ABB RobotStudio station: Station_[09.05.13]workingpinattach.rspag

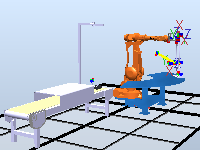
--- station ---
Station Station_[09.05.13]workingpinattach (saved by RobotStudio format 3)
Controller IRB2400_10kg_1.5m_3, task T_ROB1: task frame (RAPID world) sits at (0, 0, 226) mm in the station
Controller IRB2400_10kg_1.5m_3
  mechanical unit ROB_1: IRB2400_10_150__02, 6 joints, base frame (0, 0, -10) mm
Layout (positions relative to the parent item):
  - IRB2400_10_150__02 [mechanism, from Robots\IRB2400_10_150__02.rslib] at (0, 0, 216) mm; joint values [0, 0, 0, 0, 0, 0] (rad or m)
  - Table3_2 [part]
  - SC_RightDispenser [smart component] at (848.89, 660.39, 707) mm, rotated rx 0 ry 0 rz -142.5 deg
      signals: DI diNewPin, DO doPinInPosition2, DO doPinInPosition1
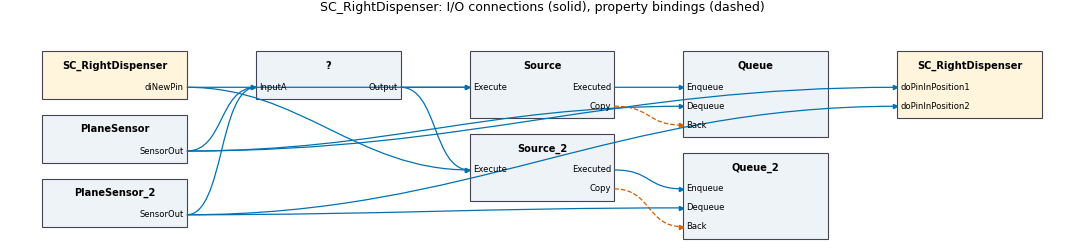
      connections:
        SC_RightDispenser.diNewPin -> Source.Execute
        Source.Executed -> Queue.Enqueue
        PlaneSensor.SensorOut -> Queue.Dequeue
        PlaneSensor.SensorOut -> SC_RightDispenser.doPinInPosition1
        PlaneSensor.SensorOut -> ?.InputA
        ?.Output -> Source.Execute
        SC_RightDispenser.diNewPin -> Source_2.Execute
        Source_2.Executed -> Queue_2.Enqueue
        PlaneSensor_2.SensorOut -> Queue_2.Dequeue
        PlaneSensor_2.SensorOut -> SC_RightDispenser.doPinInPosition2
        PlaneSensor_2.SensorOut -> ?.InputA
        ?.Output -> Source_2.Execute
        Source.Copy => Queue.Back
        Source_2.Copy => Queue_2.Back
    - Dispenser [part]
    - Source [smart component]
        properties: Source=Pin; Copy=Pin_23; Parent=(none); Position=[-0.078 0.0985 0.189]; Orientation=[0 0 0]; Transient=false
        signals: DI Execute, DO Executed
    - Queue [smart component]
        properties: Back=Pin_23; Front=(none); Queue={5aa4b278-0833-4ca9-af8d-253aa8523874};{1baac950-fc54-4ea7-852c-7f888843f6f9};{b4b16473-bd2b-40f5-a110-90fbcba822d9};{d003a69b-5307-4c56-b226-d498155ba824};{d659394f-77c7-41ee-9797-cd61472f6401};{a8294731-aa9f-4324-81a7-55ebbef1ff1c};{1eff712e-2c63-4fa8-99b0-fad1482486d3};{b15f9735-19cd-4f7a-8d4f-e540a16427f5};{02485707-3f80-4cc3-94a6-af0fe382acfb};{ec0e8ce0-b480-4ff5-b740-0a7d244ffb35};{21e78636-7eb3-4061-8dde-926c3e464303};{0772fef3-b80e-464b-9cad-322a585d167a};{d8ed8ead-e522-4938-9c7c-7997e1d5aae1};{4dfefca0-2913-4484-9455-684dfc1cbf5a};{f8c8569f-a97f-4f57-84f0-3da59c0f2755};{9fd95979-e5cf-4fa7-b177-2c560699c82c};{84f56170-3294-4345-a728-b2bfe69be833};{b3710d51-6f0f-48ac-9b0f-811ac7c7d083};{c8300349-23e3-4531-beb4-4210900096fb};{31c2e06e-432b-4cd5-8dfd-12cdd0c38bbf};{f6bc1e00-ec05-46bf-9f1a-fcc25cb6084b};{46f4262a-e9c9-45b1-8eff-bed77a1a9e5b};{07cc3b07-c3da-44db-b33b-99881492d9cc};{0c369fdb-a0e7-4beb-a0c1-abd25c6b2a43};{d9cb4cdb-12a7-4146-bf1e-65335fe6fd56};{f09a15e7-f9e4-4c16-add7-657cccb8590f};{c20793dd-1a91-48a1-8edb-9b1aca8d6d7f};{7fbcc782-7f9e-47c5-a7b7-ac04b253ef72};{f46b459a-9e88-46de-a41f-ecde2c97a1c4};{a4b9086d-e076-476d-b3ee-a23e91ee6609};{9ff53e84-8ebc-4345-9cc4-0476dc4b857f};{650503f2-9794-4bb9-bd75-77f7f6044b7b};{58395fe3-f9e1-4cbe-aa54-a35298f9d1c5};{7826030e-95bb-4bf6-b21f-9a7d91df32f4};{2942a0d1-30e6-4527-84a4-878f9b334dec};{a0ef5e72-34a5-445e-b23b-6c91bdee101a};{aa2624ab-89f7-405f-9ffa-69efbc3a4434};{9792617b-04a4-4cec-aa8d-3159fcd6b685}; NumberOfObjects=0
        signals: DI Enqueue, DI Dequeue, DI Clear, DI Delete, DI DeleteAll
    - LinearMover [smart component]
        properties: Object=Queue; Direction=[0 0 -0.07]; Speed=0.05; Reference=Global; ReferenceObject=(none)
        signals: DI Execute
    - PlaneSensor [smart component]
        properties: Origin=[-0.0530000000000006 0.1235 0.1195]; Axis1=[-0.03 0 0]; Axis2=[0 -0.04 0]; SensedPart=(none)
        signals: DI Active, DO SensorOut
      - _sensorPart_ [part]
    - Pin [part] at (-78, 98.5, 189) mm
    - Source_2 [smart component]
        properties: Source=Pin_2; Copy=Pin_2_24; Parent=(none); Position=[-0.078 -0.0985 0.198]; Orientation=[0 0 0]; Transient=false
        signals: DI Execute, DO Executed
    - Queue_2 [smart component]
        properties: Back=Pin_2_24; Front=(none); Queue={168b000f-829e-439e-a2b5-5bc5735400ce};{aacdfd62-2178-4132-b345-2cd6db76197d};{33bd895a-7dcf-445c-8a77-0a7b01e583dc};{c1a42cbc-38c3-48e5-a615-b149ac9d8780};{fcea76f5-b349-47ef-a520-1d1e9307533b};{d936eec8-07d3-4a18-b33b-be549f4009da};{161ff837-8ce6-447d-8217-59dc5e5add53};{a4db4600-beb4-451b-b75b-f36278185638};{fac26080-080b-42e5-8e31-79509598499f};{631b6ef4-884c-4e99-a73e-a0a20b005bbd};{c6922cb5-858b-4dce-bc49-d50c5bb6ff29};{df2a1232-f236-477f-a341-c0e7247ec374};{648e1593-9b95-4c8f-9a3a-4728290fef8c};{9aba8fcf-9d7f-441d-92fe-144ce1ccaea8};{d7b75440-58f5-4476-b5ce-f36666ff7cde};{5c9701ab-d039-4b3a-b377-62889d6251d5};{ccb0f00a-3f08-42c3-ae08-1f0b770d0277};{706e7c72-34ce-4f8c-bd75-a496f5af5a3b};{9b14f38f-1dc8-4293-b5b1-19b5e9014979};{c981c30e-2b93-423a-a409-ef6430437ced};{65c45e0e-b128-4bcf-862a-bd4cb12c0043};{fb18c748-94d3-4804-ba03-343ec976cce9};{90ce3d6b-e0db-4966-a4a1-dfc91785cb07};{f4c8c46d-6357-42e6-99c9-4a127ac338b9};{b14c1a72-e7b7-41f2-882c-7b7c624fc3bd};{c197bb96-9f99-45e2-aeb0-6d90c68a8177}; NumberOfObjects=0
        signals: DI Enqueue, DI Dequeue, DI Clear, DI Delete, DI DeleteAll
    - LinearMover_2 [smart component]
        properties: Object=Queue_2; Direction=[0 0 -0.07]; Speed=0.05; Reference=Global; ReferenceObject=(none)
        signals: DI Execute
    - PlaneSensor_2 [smart component]
        properties: Origin=[-0.053 -0.1235 0.1195]; Axis1=[-0.03 0 0]; Axis2=[0 0.04 0]; SensedPart=(none)
        signals: DI Active, DO SensorOut
      - _sensorPart_ [part]
    - Pin_2 [part] at (-78, -98.5, 189) mm
    - Pin_23 [part] at (2071.41, 800.68, -37.38) mm, rotated rx -0.03 ry 0 rz -128.08 deg
    - Pin_2_24 [part] at (1981.85, 913.72, -36.32) mm, rotated rx -0.03 ry 0.01 rz -128.09 deg
  - NewSmartGripper[040513] [smart component] at (940, 0, 1671) mm, rotated rx 0 ry 90 rz 0 deg
      signals: DO doPinAttached, DI diAttachPin, DO doPalletAttached, DO doGripperTouchesTable
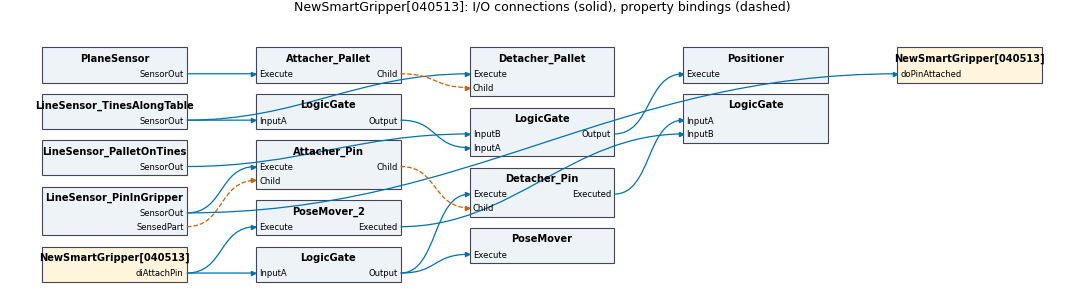
      connections:
        PlaneSensor.SensorOut -> Attacher_Pallet.Execute
        LineSensor_TinesAlongTable.SensorOut -> Detacher_Pallet.Execute
        LineSensor_TinesAlongTable.SensorOut -> LogicGate.InputA
        LineSensor_PalletOnTines.SensorOut -> LogicGate.InputB
        LogicGate.Output -> LogicGate.InputA
        LogicGate.Output -> Positioner.Execute
        LineSensor_PinInGripper.SensorOut -> Attacher_Pin.Execute
        LineSensor_PinInGripper.SensorOut -> NewSmartGripper[040513].doPinAttached
        NewSmartGripper[040513].diAttachPin -> PoseMover_2.Execute
        NewSmartGripper[040513].diAttachPin -> LogicGate.InputA
        Detacher_Pin.Executed -> LogicGate.InputA
        PoseMover_2.Executed -> LogicGate.InputB
        LogicGate.Output -> PoseMover.Execute
        LogicGate.Output -> Detacher_Pin.Execute
        Attacher_Pallet.Child => Detacher_Pallet.Child
        Attacher_Pin.Child => Detacher_Pin.Child
        LineSensor_PinInGripper.SensedPart => Attacher_Pin.Child
    - LineSensor_PinInGripper [smart component, from Libraries\LineSensor.rslib]
        properties: Start=[0.03 0 0.1702]; End=[0.03 0 0.16]; Radius=0.002; SensedPart=(none); SensedPoint=[0 0 0]
      - _sensorPart_ [part]
    - LineSensor_PalletOnTines [smart component, from Libraries\LineSensor.rslib]
        properties: Start=[-0.109 0.07175 0.233]; End=[-0.109 0.07175 0.23]; Radius=0.0012; SensedPart=(none); SensedPoint=[0 0 0]
      - _sensorPart_ [part]
    - LineSensor_TinesAlongTable [smart component, from Libraries\LineSensor.rslib]
        properties: Start=[-0.15 0.15 0]; End=[-0.12 0.15 0]; Radius=0.004; SensedPart=(none); SensedPoint=[0 0 0]
      - _sensorPart_ [part]
    - PoseMover [smart component, from Libraries\PoseMover.rslib]
        properties: Mechanism=NewGripperMech; Pose=3; Duration=0.2
    - PoseMover_2 [smart component, from Libraries\PoseMover.rslib]
        properties: Mechanism=NewGripperMech; Pose=2; Duration=0.2
    - NewGripperMech [mechanism] at (0, 0, 0) mm; joint values [-0.008, 0.008] (rad or m)
        TCP tTine at (-114.5, 0, 234.15) mm, rotated rx 0 ry 0 rz 180 deg
        TCP tGrip at (30, 0, 180) mm, rotated rx 0 ry -90 rz 0 deg
        links: L1, L2, L3
    - LogicSRLatchPalletAttached [smart component, from Libraries\LogicSRLatch.rslib]
    - PlaneSensor [smart component, from Libraries\PlaneSensor.rslib]
        properties: Origin=[-0.1 -0.05 0.055]; Axis1=[0.02 0 0]; Axis2=[0 0.1 0]; SensedPart=(none)
      - _sensorPart_ [part]
    - LinearMover [smart component, from Libraries\LinearMover.rslib]
        properties: Object=Pallet; Direction=[0 0 -0.01]; Speed=0.1; Reference=Object; ReferenceObject=PlaneSensor
    - Positioner [smart component, from Libraries\Positioner.rslib]
        properties: Object=Pallet; Position=[-0.143 -0.11 0.273]; Orientation=[0 1.5707963267949 0]; Reference=Object; ReferenceObject=PlaneSensor
    - Attacher_Pallet [smart component, from Libraries\Attacher.rslib]
        properties: Parent=NewSmartGripper[040513]; Flange=0; Child=Pallet; Mount=false; Offset=[0 0 0]; Orientation=[0 0 0]
    - LinearMover_stop [smart component, from Libraries\LinearMover.rslib]
        properties: Object=Pallet; Direction=[0 0 1E-07]; Speed=1E-07; Reference=Object; ReferenceObject=PlaneSensor
    - Detacher_Pallet [smart component, from Libraries\Detacher.rslib]
        properties: Child=Pallet; KeepPosition=true
    - LogicGate [smart component, from Libraries\LogicGate.rslib]
        properties: Operator=NOT; Delay=0
    - LogicGate [smart component, from Libraries\LogicGate.rslib]
        properties: Operator=AND; Delay=0
    - Attacher_Pin [smart component, from Libraries\Attacher_1.rslib]
        properties: Parent=NewSmartGripper[040513]; Flange=0; Child=(none); Mount=false; Offset=[0 0 0]; Orientation=[0 0 0]
    - Detacher_Pin [smart component, from Libraries\Detacher.rslib]
        properties: Child=(none); KeepPosition=true
    - LogicGate [smart component, from Libraries\LogicGate.rslib]
        properties: Operator=AND; Delay=0
    - LogicGate [smart component, from Libraries\LogicGate.rslib]
        properties: Operator=NOT; Delay=0
  - SC_Conveyor[190413] [smart component] at (45.5, -3634, 0) mm
      signals: DI diPalletOut, DI diPalletIn, DO doPalletAtEnd, DO doPalletAtStart, DO diPalletMovingOut, DO doPalletMovingIn, DI diConDir, DI diConRun
      connections:
        PlaneSensor_Start.SensorOut -> PalletOnConANDdiPalletOut.InputA
        PlaneSensor_Start.SensorOut -> SC_Conveyor[190413].doPalletAtStart
        SC_Conveyor[190413].diPalletOut -> PalletOnConANDdiPalletOut.InputB
        SC_Conveyor[190413].diPalletIn -> PalletOnConANDdiPalletIn.InputB
        PalletOnConANDdiPalletOut.Output -> LinearMoverOut.Execute
        PalletOnConANDdiPalletOut.Output -> SC_Conveyor[190413].diPalletMovingOut
        PlaneSensor_End.SensorOut -> PalletOnConANDdiPalletIn.InputA
        PlaneSensor_End.SensorOut -> SC_Conveyor[190413].doPalletAtEnd
        PalletOnConANDdiPalletIn.Output -> LinearMover_In.Execute
        PalletOnConANDdiPalletIn.Output -> SC_Conveyor[190413].doPalletMovingIn
        PlaneSensor_Start.SensedPart => LinearMoverOut.Object
        PlaneSensor_End.SensedPart => LinearMover_In.Object
    - Conveyor3 [part] at (0, 0, 606) mm
    - PlaneSensor_Start [smart component]
        properties: Origin=[-0.05 0.4 0.62]; Axis1=[-0.5 0 0]; Axis2=[0 2.1 0]; SensedPart=Pallet
        signals: DI Active, DO SensorOut
      - _sensorPart_ [part]
    - PlaneSensor_End [smart component]
        properties: Origin=[-0.05 0 0.62]; Axis1=[-0.5 0 0]; Axis2=[0 2.2 0]; SensedPart=(none)
        signals: DI Active, DO SensorOut
      - _sensorPart_ [part]
    - LinearMoverOut [smart component]
        properties: Object=Pallet; Direction=[0 -1 0]; Speed=0.6; Reference=Global; ReferenceObject=(none)
        signals: DI Execute
    - LinearMover_In [smart component]
        properties: Object=(none); Direction=[0 1 0]; Speed=0.6; Reference=Global; ReferenceObject=(none)
        signals: DI Execute
    - LogicSRLatchOut [smart component]
        signals: DI Set, DI Reset, DO Output, DO InvOutput
    - LogicSRLatchIn [smart component]
        signals: DI Set, DI Reset, DO Output, DO InvOutput
    - PalletOnConANDdiPalletOut [smart component, from Libraries\LogicGate.rslib]
        properties: Operator=AND; Delay=0
    - PalletOnConANDdiPalletIn [smart component, from Libraries\LogicGate.rslib]
        properties: Operator=AND; Delay=0
    - Attatcher_PinInPallet [smart component, from Libraries\Attacher_1.rslib]
        properties: Parent=Pallet; Flange=0; Child=(none); Mount=false; Offset=[0 0 0]; Orientation=[0 0 0]
  - PalletSmartComponent [smart component] at (-124.56, -1382.89, 612.85) mm
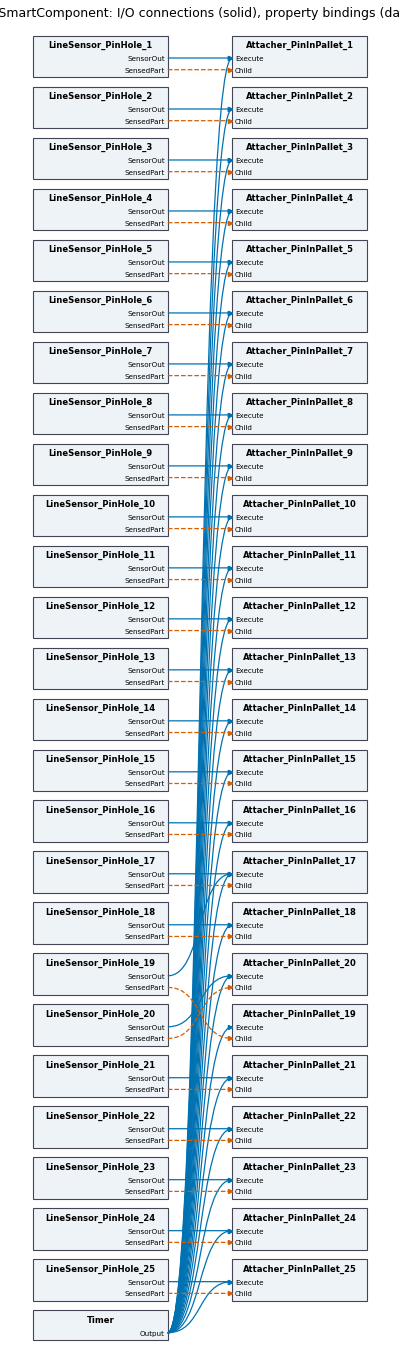
      connections:
        LineSensor_PinHole_1.SensorOut -> Attacher_PinInPallet_1.Execute
        LineSensor_PinHole_2.SensorOut -> Attacher_PinInPallet_2.Execute
        LineSensor_PinHole_3.SensorOut -> Attacher_PinInPallet_3.Execute
        LineSensor_PinHole_4.SensorOut -> Attacher_PinInPallet_4.Execute
        LineSensor_PinHole_5.SensorOut -> Attacher_PinInPallet_5.Execute
        LineSensor_PinHole_6.SensorOut -> Attacher_PinInPallet_6.Execute
        LineSensor_PinHole_7.SensorOut -> Attacher_PinInPallet_7.Execute
        LineSensor_PinHole_8.SensorOut -> Attacher_PinInPallet_8.Execute
        LineSensor_PinHole_9.SensorOut -> Attacher_PinInPallet_9.Execute
        LineSensor_PinHole_10.SensorOut -> Attacher_PinInPallet_10.Execute
        LineSensor_PinHole_11.SensorOut -> Attacher_PinInPallet_11.Execute
        LineSensor_PinHole_12.SensorOut -> Attacher_PinInPallet_12.Execute
        LineSensor_PinHole_13.SensorOut -> Attacher_PinInPallet_13.Execute
        LineSensor_PinHole_14.SensorOut -> Attacher_PinInPallet_14.Execute
        LineSensor_PinHole_15.SensorOut -> Attacher_PinInPallet_15.Execute
        LineSensor_PinHole_16.SensorOut -> Attacher_PinInPallet_16.Execute
        LineSensor_PinHole_17.SensorOut -> Attacher_PinInPallet_17.Execute
        LineSensor_PinHole_18.SensorOut -> Attacher_PinInPallet_18.Execute
        LineSensor_PinHole_19.SensorOut -> Attacher_PinInPallet_17.Execute
        LineSensor_PinHole_20.SensorOut -> Attacher_PinInPallet_20.Execute
        LineSensor_PinHole_21.SensorOut -> Attacher_PinInPallet_21.Execute
        LineSensor_PinHole_22.SensorOut -> Attacher_PinInPallet_22.Execute
        LineSensor_PinHole_23.SensorOut -> Attacher_PinInPallet_23.Execute
        LineSensor_PinHole_24.SensorOut -> Attacher_PinInPallet_24.Execute
        LineSensor_PinHole_25.SensorOut -> Attacher_PinInPallet_25.Execute
        Timer.Output -> Attacher_PinInPallet_1.Execute
        Timer.Output -> Attacher_PinInPallet_2.Execute
        Timer.Output -> Attacher_PinInPallet_3.Execute
        Timer.Output -> Attacher_PinInPallet_4.Execute
        Timer.Output -> Attacher_PinInPallet_5.Execute
        Timer.Output -> Attacher_PinInPallet_6.Execute
        Timer.Output -> Attacher_PinInPallet_7.Execute
        Timer.Output -> Attacher_PinInPallet_8.Execute
        Timer.Output -> Attacher_PinInPallet_9.Execute
        Timer.Output -> Attacher_PinInPallet_25.Execute
        Timer.Output -> Attacher_PinInPallet_24.Execute
        Timer.Output -> Attacher_PinInPallet_23.Execute
        Timer.Output -> Attacher_PinInPallet_22.Execute
        Timer.Output -> Attacher_PinInPallet_21.Execute
        Timer.Output -> Attacher_PinInPallet_20.Execute
        Timer.Output -> Attacher_PinInPallet_19.Execute
        Timer.Output -> Attacher_PinInPallet_18.Execute
        Timer.Output -> Attacher_PinInPallet_17.Execute
        Timer.Output -> Attacher_PinInPallet_16.Execute
        Timer.Output -> Attacher_PinInPallet_15.Execute
        Timer.Output -> Attacher_PinInPallet_14.Execute
        Timer.Output -> Attacher_PinInPallet_13.Execute
        Timer.Output -> Attacher_PinInPallet_12.Execute
        Timer.Output -> Attacher_PinInPallet_11.Execute
        Timer.Output -> Attacher_PinInPallet_10.Execute
        LineSensor_PinHole_1.SensedPart => Attacher_PinInPallet_1.Child
        LineSensor_PinHole_2.SensedPart => Attacher_PinInPallet_2.Child
        LineSensor_PinHole_3.SensedPart => Attacher_PinInPallet_3.Child
        LineSensor_PinHole_4.SensedPart => Attacher_PinInPallet_4.Child
        LineSensor_PinHole_5.SensedPart => Attacher_PinInPallet_5.Child
        LineSensor_PinHole_6.SensedPart => Attacher_PinInPallet_6.Child
        LineSensor_PinHole_7.SensedPart => Attacher_PinInPallet_7.Child
        LineSensor_PinHole_8.SensedPart => Attacher_PinInPallet_8.Child
        LineSensor_PinHole_9.SensedPart => Attacher_PinInPallet_9.Child
        LineSensor_PinHole_10.SensedPart => Attacher_PinInPallet_10.Child
        LineSensor_PinHole_12.SensedPart => Attacher_PinInPallet_12.Child
        LineSensor_PinHole_11.SensedPart => Attacher_PinInPallet_11.Child
        LineSensor_PinHole_13.SensedPart => Attacher_PinInPallet_13.Child
        LineSensor_PinHole_14.SensedPart => Attacher_PinInPallet_14.Child
        LineSensor_PinHole_15.SensedPart => Attacher_PinInPallet_15.Child
        LineSensor_PinHole_16.SensedPart => Attacher_PinInPallet_16.Child
        LineSensor_PinHole_17.SensedPart => Attacher_PinInPallet_17.Child
        LineSensor_PinHole_18.SensedPart => Attacher_PinInPallet_18.Child
        LineSensor_PinHole_20.SensedPart => Attacher_PinInPallet_20.Child
        LineSensor_PinHole_21.SensedPart => Attacher_PinInPallet_21.Child
        LineSensor_PinHole_22.SensedPart => Attacher_PinInPallet_22.Child
        LineSensor_PinHole_23.SensedPart => Attacher_PinInPallet_23.Child
        LineSensor_PinHole_19.SensedPart => Attacher_PinInPallet_19.Child
        LineSensor_PinHole_24.SensedPart => Attacher_PinInPallet_24.Child
        LineSensor_PinHole_25.SensedPart => Attacher_PinInPallet_25.Child
    - Pallet [part] at (0, 0, 0) mm, rotated rx 0 ry 0 rz 89.99 deg
    - Attacher_PinInPallet_1 [smart component, from Libraries\Attacher_1.rslib]
        properties: Parent=Pallet; Flange=0; Child=(none); Mount=false; Offset=[0 0 0]; Orientation=[0 0 0]
    - PlaneSensor [smart component, from Libraries\PlaneSensor_1.rslib] at (-200, 27, 65) mm
        properties: Origin=[0 0 -0.008]; Axis1=[0.17 0 0]; Axis2=[0 0.17 0]; SensedPart=Pallet
      - _sensorPart_ [part]
    - LineSensor_PinHole_1 [smart component, from Libraries\LineSensor_1.rslib] at (-180.75, 40.67, 37.99) mm
        properties: Start=[0 0 0.001]; End=[0 0 0.02]; Radius=0; SensedPart=(none); SensedPoint=[0 0 0]
      - _sensorPart_ [part]
    - LineSensor_PinHole_2 [smart component, from Libraries\LineSensor_1.rslib] at (-180.75, 75.67, 37.99) mm
        properties: Start=[0 0 0.001]; End=[0 0 0.02]; Radius=0; SensedPart=(none); SensedPoint=[0 0 0]
      - _sensorPart_ [part]
    - LineSensor_PinHole_3 [smart component, from Libraries\LineSensor_1.rslib] at (-180.75, 110.67, 37.99) mm
        properties: Start=[0 0 0.001]; End=[0 0 0.02]; Radius=0; SensedPart=(none); SensedPoint=[0 0 0]
      - _sensorPart_ [part]
    - LineSensor_PinHole_4 [smart component, from Libraries\LineSensor_1.rslib] at (-180.75, 145.67, 37.99) mm
        properties: Start=[0 0 0.001]; End=[0 0 0.02]; Radius=0; SensedPart=Pin_23; SensedPoint=[-0.305319030761719 -1.2372265625 0.669619873046875]
      - _sensorPart_ [part]
    - LineSensor_PinHole_5 [smart component, from Libraries\LineSensor_1.rslib] at (-180.75, 180.67, 37.99) mm
        properties: Start=[0 0 0.001]; End=[0 0 0.02]; Radius=0; SensedPart=(none); SensedPoint=[0 0 0]
      - _sensorPart_ [part]
    - LineSensor_PinHole_6 [smart component, from Libraries\LineSensor_1.rslib] at (-145.75, 40.67, 37.99) mm
        properties: Start=[0 0 0.001]; End=[0 0 0.02]; Radius=0; SensedPart=(none); SensedPoint=[0 0 0]
      - _sensorPart_ [part]
    - LineSensor_PinHole_7 [smart component, from Libraries\LineSensor_1.rslib] at (-145.75, 75.67, 37.99) mm
        properties: Start=[0 0 0.001]; End=[0 0 0.02]; Radius=0; SensedPart=(none); SensedPoint=[0 0 0]
      - _sensorPart_ [part]
    - LineSensor_PinHole_8 [smart component, from Libraries\LineSensor_1.rslib] at (-145.75, 110.67, 37.99) mm
        properties: Start=[0 0 0.001]; End=[0 0 0.02]; Radius=0; SensedPart=(none); SensedPoint=[0 0 0]
      - _sensorPart_ [part]
    - LineSensor_PinHole_9 [smart component, from Libraries\LineSensor_1.rslib] at (-145.75, 145.67, 37.99) mm
        properties: Start=[0 0 0.001]; End=[0 0 0.02]; Radius=0; SensedPart=(none); SensedPoint=[0 0 0]
      - _sensorPart_ [part]
    - LineSensor_PinHole_10 [smart component, from Libraries\LineSensor_1.rslib] at (-145.75, 180.67, 37.99) mm
        properties: Start=[0 0 0.001]; End=[0 0 0.02]; Radius=0; SensedPart=(none); SensedPoint=[0 0 0]
      - _sensorPart_ [part]
    - LineSensor_PinHole_11 [smart component, from Libraries\LineSensor_1.rslib] at (-110.75, 40.67, 37.99) mm
        properties: Start=[0 0 0.001]; End=[0 0 0.02]; Radius=0; SensedPart=(none); SensedPoint=[0 0 0]
      - _sensorPart_ [part]
    - LineSensor_PinHole_12 [smart component, from Libraries\LineSensor_1.rslib] at (-110.75, 75.67, 37.99) mm
        properties: Start=[0 0 0.001]; End=[0 0 0.02]; Radius=0; SensedPart=(none); SensedPoint=[0 0 0]
      - _sensorPart_ [part]
    - LineSensor_PinHole_13 [smart component, from Libraries\LineSensor_1.rslib] at (-110.75, 110.67, 37.99) mm
        properties: Start=[0 0 0.001]; End=[0 0 0.02]; Radius=0; SensedPart=(none); SensedPoint=[0 0 0]
      - _sensorPart_ [part]
    - LineSensor_PinHole_14 [smart component, from Libraries\LineSensor_1.rslib] at (-110.75, 145.67, 37.99) mm
        properties: Start=[0 0 0.001]; End=[0 0 0.02]; Radius=0; SensedPart=(none); SensedPoint=[0 0 0]
      - _sensorPart_ [part]
    - LineSensor_PinHole_15 [smart component, from Libraries\LineSensor_1.rslib] at (-110.75, 180.67, 37.99) mm
        properties: Start=[0 0 0.001]; End=[0 0 0.02]; Radius=0; SensedPart=(none); SensedPoint=[0 0 0]
      - _sensorPart_ [part]
    - LineSensor_PinHole_16 [smart component, from Libraries\LineSensor_1.rslib] at (-75.75, 40.67, 37.99) mm
        properties: Start=[0 0 0.001]; End=[0 0 0.02]; Radius=0; SensedPart=(none); SensedPoint=[0 0 0]
      - _sensorPart_ [part]
    - LineSensor_PinHole_17 [smart component, from Libraries\LineSensor_1.rslib] at (-75.75, 75.67, 37.99) mm
        properties: Start=[0 0 0.001]; End=[0 0 0.02]; Radius=0; SensedPart=(none); SensedPoint=[0 0 0]
      - _sensorPart_ [part]
    - LineSensor_PinHole_18 [smart component, from Libraries\LineSensor_1.rslib] at (-75.75, 110.67, 37.99) mm
        properties: Start=[0 0 0.001]; End=[0 0 0.02]; Radius=0; SensedPart=(none); SensedPoint=[0 0 0]
      - _sensorPart_ [part]
    - LineSensor_PinHole_19 [smart component, from Libraries\LineSensor_1.rslib] at (-75.75, 145.67, 37.99) mm
        properties: Start=[0 0 0.001]; End=[0 0 0.02]; Radius=0; SensedPart=(none); SensedPoint=[0 0 0]
      - _sensorPart_ [part]
    - LineSensor_PinHole_20 [smart component, from Libraries\LineSensor_1.rslib] at (-75.75, 180.67, 37.99) mm
        properties: Start=[0 0 0.001]; End=[0 0 0.02]; Radius=0; SensedPart=(none); SensedPoint=[0 0 0]
      - _sensorPart_ [part]
    - LineSensor_PinHole_21 [smart component, from Libraries\LineSensor_1.rslib] at (-40.75, 40.67, 37.99) mm
        properties: Start=[0 0 0.001]; End=[0 0 0.02]; Radius=0; SensedPart=(none); SensedPoint=[0 0 0]
      - _sensorPart_ [part]
    - LineSensor_PinHole_22 [smart component, from Libraries\LineSensor_1.rslib] at (-40.75, 75.67, 37.99) mm
        properties: Start=[0 0 0.001]; End=[0 0 0.02]; Radius=0; SensedPart=(none); SensedPoint=[0 0 0]
      - _sensorPart_ [part]
    - LineSensor_PinHole_23 [smart component, from Libraries\LineSensor_1.rslib] at (-40.75, 110.67, 37.99) mm
        properties: Start=[0 0 0.001]; End=[0 0 0.02]; Radius=0; SensedPart=Pin_2_24; SensedPoint=[-0.16531901550293 -1.27222644042969 0.67068212890625]
      - _sensorPart_ [part]
    - LineSensor_PinHole_24 [smart component, from Libraries\LineSensor_1.rslib] at (-40.75, 145.67, 37.99) mm
        properties: Start=[0 0 0.001]; End=[0 0 0.02]; Radius=0; SensedPart=(none); SensedPoint=[0 0 0]
      - _sensorPart_ [part]
    - LineSensor_PinHole_25 [smart component, from Libraries\LineSensor_1.rslib] at (-40.75, 180.67, 37.99) mm
        properties: Start=[0 0 0.001]; End=[0 0 0.02]; Radius=0; SensedPart=(none); SensedPoint=[0 0 0]
      - _sensorPart_ [part]
    - Attacher_PinInPallet_2 [smart component, from Libraries\Attacher_1.rslib]
        properties: Parent=Pallet; Flange=0; Child=(none); Mount=false; Offset=[0 0 0]; Orientation=[0 0 0]
    - Attacher_PinInPallet_3 [smart component, from Libraries\Attacher_1.rslib]
        properties: Parent=Pallet; Flange=0; Child=(none); Mount=false; Offset=[0 0 0]; Orientation=[0 0 0]
    - Attacher_PinInPallet_4 [smart component, from Libraries\Attacher_1.rslib]
        properties: Parent=Pallet; Flange=0; Child=Pin_23; Mount=false; Offset=[0 0 0]; Orientation=[0 0 0]
    - Attacher_PinInPallet_5 [smart component, from Libraries\Attacher_1.rslib]
        properties: Parent=Pallet; Flange=0; Child=(none); Mount=false; Offset=[0 0 0]; Orientation=[0 0 0]
    - Attacher_PinInPallet_6 [smart component, from Libraries\Attacher_1.rslib]
        properties: Parent=Pallet; Flange=0; Child=(none); Mount=false; Offset=[0 0 0]; Orientation=[0 0 0]
    - Attacher_PinInPallet_7 [smart component, from Libraries\Attacher_1.rslib]
        properties: Parent=Pallet; Flange=0; Child=(none); Mount=false; Offset=[0 0 0]; Orientation=[0 0 0]
    - Attacher_PinInPallet_8 [smart component, from Libraries\Attacher_1.rslib]
        properties: Parent=Pallet; Flange=0; Child=(none); Mount=false; Offset=[0 0 0]; Orientation=[0 0 0]
    - Attacher_PinInPallet_9 [smart component, from Libraries\Attacher_1.rslib]
        properties: Parent=Pallet; Flange=0; Child=(none); Mount=false; Offset=[0 0 0]; Orientation=[0 0 0]
    - Attacher_PinInPallet_10 [smart component, from Libraries\Attacher_1.rslib]
        properties: Parent=Pallet; Flange=0; Child=(none); Mount=false; Offset=[0 0 0]; Orientation=[0 0 0]
    - Attacher_PinInPallet_11 [smart component, from Libraries\Attacher_1.rslib]
        properties: Parent=Pallet; Flange=0; Child=(none); Mount=false; Offset=[0 0 0]; Orientation=[0 0 0]
    - Attacher_PinInPallet_12 [smart component, from Libraries\Attacher_1.rslib]
        properties: Parent=Pallet; Flange=0; Child=(none); Mount=false; Offset=[0 0 0]; Orientation=[0 0 0]
    - Attacher_PinInPallet_13 [smart component, from Libraries\Attacher_1.rslib]
        properties: Parent=Pallet; Flange=0; Child=(none); Mount=false; Offset=[0 0 0]; Orientation=[0 0 0]
    - Attacher_PinInPallet_14 [smart component, from Libraries\Attacher_1.rslib]
        properties: Parent=Pallet; Flange=0; Child=(none); Mount=false; Offset=[0 0 0]; Orientation=[0 0 0]
    - Attacher_PinInPallet_15 [smart component, from Libraries\Attacher_1.rslib]
        properties: Parent=Pallet; Flange=0; Child=(none); Mount=false; Offset=[0 0 0]; Orientation=[0 0 0]
    - Attacher_PinInPallet_16 [smart component, from Libraries\Attacher_1.rslib]
        properties: Parent=Pallet; Flange=0; Child=(none); Mount=false; Offset=[0 0 0]; Orientation=[0 0 0]
    - Attacher_PinInPallet_17 [smart component, from Libraries\Attacher_1.rslib]
        properties: Parent=Pallet; Flange=0; Child=(none); Mount=false; Offset=[0 0 0]; Orientation=[0 0 0]
    - Attacher_PinInPallet_18 [smart component, from Libraries\Attacher_1.rslib]
        properties: Parent=Pallet; Flange=0; Child=(none); Mount=false; Offset=[0 0 0]; Orientation=[0 0 0]
    - Attacher_PinInPallet_19 [smart component, from Libraries\Attacher_1.rslib]
        properties: Parent=Pallet; Flange=0; Child=(none); Mount=false; Offset=[0 0 0]; Orientation=[0 0 0]
    - Attacher_PinInPallet_20 [smart component, from Libraries\Attacher_1.rslib]
        properties: Parent=Pallet; Flange=0; Child=(none); Mount=false; Offset=[0 0 0]; Orientation=[0 0 0]
    - Attacher_PinInPallet_21 [smart component, from Libraries\Attacher_1.rslib]
        properties: Parent=Pallet; Flange=0; Child=(none); Mount=false; Offset=[0 0 0]; Orientation=[0 0 0]
    - Attacher_PinInPallet_22 [smart component, from Libraries\Attacher_1.rslib]
        properties: Parent=Pallet; Flange=0; Child=(none); Mount=false; Offset=[0 0 0]; Orientation=[0 0 0]
    - Attacher_PinInPallet_23 [smart component, from Libraries\Attacher_1.rslib]
        properties: Parent=Pallet; Flange=0; Child=Pin_2_24; Mount=false; Offset=[0 0 0]; Orientation=[0 0 0]
    - Attacher_PinInPallet_24 [smart component, from Libraries\Attacher_1.rslib]
        properties: Parent=Pallet; Flange=0; Child=(none); Mount=false; Offset=[0 0 0]; Orientation=[0 0 0]
    - Attacher_PinInPallet_25 [smart component, from Libraries\Attacher_1.rslib]
        properties: Parent=Pallet; Flange=0; Child=(none); Mount=false; Offset=[0 0 0]; Orientation=[0 0 0]
    - Timer [smart component, from Libraries\Timer.rslib]
        properties: StartTime=0; Interval=1; Repeat=true; CurrentTime=104.472
  - Frame_1 [frame] at (710.04, 677.11, 1017.54) mm, rotated rx -135.34 ry 89.95 rz -97.28 deg
Attachment: NewSmartGripper[040513] is attached to IRB2400_10_150__02 / Link6
Attachment: PlaneSensor is attached to Pallet
Attachment: LineSensor_PinHole_1 is attached to Pallet
Attachment: LineSensor_PinHole_2 is attached to Pallet
Attachment: LineSensor_PinHole_3 is attached to Pallet
Attachment: LineSensor_PinHole_4 is attached to Pallet
Attachment: LineSensor_PinHole_5 is attached to Pallet
Attachment: LineSensor_PinHole_6 is attached to Pallet
Attachment: LineSensor_PinHole_7 is attached to Pallet
Attachment: LineSensor_PinHole_8 is attached to Pallet
Attachment: LineSensor_PinHole_9 is attached to Pallet
Attachment: LineSensor_PinHole_10 is attached to Pallet
Attachment: LineSensor_PinHole_11 is attached to Pallet
Attachment: LineSensor_PinHole_12 is attached to Pallet
Attachment: LineSensor_PinHole_13 is attached to Pallet
Attachment: LineSensor_PinHole_14 is attached to Pallet
Attachment: LineSensor_PinHole_15 is attached to Pallet
Attachment: LineSensor_PinHole_16 is attached to Pallet
Attachment: LineSensor_PinHole_17 is attached to Pallet
Attachment: LineSensor_PinHole_18 is attached to Pallet
Attachment: LineSensor_PinHole_19 is attached to Pallet
Attachment: LineSensor_PinHole_20 is attached to Pallet
Attachment: LineSensor_PinHole_21 is attached to Pallet
Attachment: LineSensor_PinHole_22 is attached to Pallet
Attachment: LineSensor_PinHole_23 is attached to Pallet
Attachment: LineSensor_PinHole_24 is attached to Pallet
Attachment: LineSensor_PinHole_25 is attached to Pallet
Attachment: Pin_23 is attached to Pallet
Attachment: Pin_2_24 is attached to Pallet
EventTableEntry 5: Group=, Trigger=Grip 6, Actions=[diGRIP 7], Comment=, ActivationMode=2, Cyclic=false
EventTableTriggerIO 6: IOValue=[1], IRC5Controller=? -1, Operator=0, SignalSource=IRB2400_10kg_1.5m_3 486
EventTableActionIO 7: IOValue=[0], IRC5Controller=? -1, SignalTarget=Station_[09.05.13]workingpinattach 1
EventTableEntry 8: Group=, Trigger=Grip 9, Actions=[diGRIP 10], Comment=, ActivationMode=2, Cyclic=false
EventTableTriggerIO 9: IOValue=[0], IRC5Controller=? -1, Operator=0, SignalSource=IRB2400_10kg_1.5m_3 486
EventTableActionIO 10: IOValue=[1], IRC5Controller=? -1, SignalTarget=Station_[09.05.13]workingpinattach 1
EventTableTriggerIO 1726: IOValue=[1], IRC5Controller=? -1, Operator=0, SignalSource=IRB2400_10kg_1.5m_3 486
EventTableTriggerIO 1727: IOValue=[0], IRC5Controller=? -1, Operator=0, SignalSource=IRB2400_10kg_1.5m_3 486
EventTableEntry 1775: Group=, Trigger=ConRun 1776, Actions=[diStationConRun 1777], Comment=, ActivationMode=2, Cyclic=false
EventTableTriggerIO 1776: IOValue=[1], IRC5Controller=? -1, Operator=0, SignalSource=IRB2400_10kg_1.5m_3 486
EventTableActionIO 1777: IOValue=[1], IRC5Controller=? -1, SignalTarget=Station_[09.05.13]workingpinattach 1
EventTableEntry 1778: Group=, Trigger=ConDir 1779, Actions=[diStationConDir 1780], Comment=, ActivationMode=2, Cyclic=false
EventTableTriggerIO 1779: IOValue=[1], IRC5Controller=? -1, Operator=0, SignalSource=IRB2400_10kg_1.5m_3 486
EventTableActionIO 1780: IOValue=[1], IRC5Controller=? -1, SignalTarget=Station_[09.05.13]workingpinattach 1
EventTableEntry 1781: Group=, Trigger=ConRun 1782, Actions=[diStationConRun 1783], Comment=, ActivationMode=2, Cyclic=false
EventTableTriggerIO 1782: IOValue=[0], IRC5Controller=? -1, Operator=0, SignalSource=IRB2400_10kg_1.5m_3 486
EventTableActionIO 1783: IOValue=[0], IRC5Controller=? -1, SignalTarget=Station_[09.05.13]workingpinattach 1
EventTableEntry 1784: Group=, Trigger=ConDir 1785, Actions=[diStationConDir 1786], Comment=, ActivationMode=2, Cyclic=false
EventTableTriggerIO 1785: IOValue=[0], IRC5Controller=? -1, Operator=0, SignalSource=IRB2400_10kg_1.5m_3 486
EventTableActionIO 1786: IOValue=[0], IRC5Controller=? -1, SignalTarget=Station_[09.05.13]workingpinattach 1
Collision set CollisionSet_1:  against , near miss 0 m
Station signals: DI diRunConOUT, DI diRunConIN, DI diGRIP, DI diNewPinINDISP, DI diStationConRun, DI diStationConDir
Station logic (signal -> signal, property => property):
  Station_[09.05.13]workingpinattach.diGRIP -> NewSmartGripper[040513].diAttachPin
  Station_[09.05.13]workingpinattach.diNewPinINDISP -> SC_RightDispenser.diNewPin
  Station_[09.05.13]workingpinattach.diStationConRun -> SC_Conveyor[190413].diConRun
  Station_[09.05.13]workingpinattach.diStationConDir -> SC_Conveyor[190413].diConDir
Targets, tools, work objects and paths stored in the station and not in the controller backup, written as RAPID:
! task T_ROB1
MODULE MW
  PROC PlacePin()
    MoveJ pSlugDispG1Safe,v500,fine,tGrip;
    MoveL pSlugDispG1,v200,fine,tGrip;
    Set Grip;
    WaitTime 1;
    MoveL pSlugDispG1Safe,v200,fine,tGrip;
    MoveJ pSlugDispG2Safe,v1000,fine,tGrip;
    MoveL pSlugDispG2,v200,fine,tGrip;
    Set Grip;
    WaitTime 1;
    MoveL pSlugDispG2Safe,v200,fine,tGrip;
    MoveJ pDispConvInt,v1000,fine,tGrip;
    MoveJ Offs(pSlugPallConvCD,0,0,200),v1000,fine,tGrip;
    MoveL Offs(pSlugPallH1D, xoffset, yoffset, 50),v200,fine,tGrip;
    MoveL Offs(pSlugPallH1D, xoffset, yoffset, 0),v200,fine,tGrip;
    Reset Grip;
    WaitTime 1;
    MoveL Offs(pSlugPallH1D, xoffset, yoffset, 100),v200,fine,tGrip;
    MoveAbsJ jtCalibPos,v1000,fine,tTine;
  ENDPROC
ENDMODULE

! task T_ROB1
MODULE CalibData
  PERS tooldata Tooldata_1:=[TRUE,[[20,0,175.76],[0.707106781,0,-0.707106781,0]],[1,[0,0,1],[1,0,0,0],0,0,0]];
  PERS tooldata Tooldata_2:=[TRUE,[[-83.5,0,233],[0,0.707106781,0,0.707106781]],[1,[0,0,1],[1,0,0,0],0,0,0]];
ENDMODULE


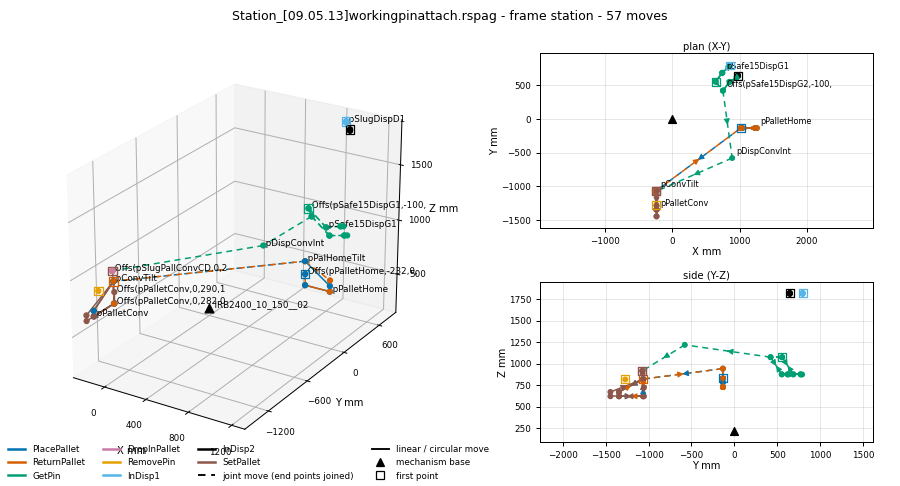
[picture p0: tool path of Station_[09.05.13]workingpinattach.rspag in frame station, 57 of 72 moves have a stored position in this frame; points joined in program order, loops and branches not executed]
--- Backups/IRB2400_10kg_1.5m_3/RAPID/TASK1/PROGMOD/CalibData.mod ---
MODULE CalibData
	PERS tooldata My_Mechanism_1:=[TRUE,[[20,0,175.76],[0.707106781,0,-0.707106781,0]],[1,[0,0,1],[1,0,0,0],0,0,0]];
	PERS tooldata My_Mechanism_2:=[TRUE,[[-83.5,0,233],[0,0.707106781,0,0.707106781]],[1,[0,0,1],[1,0,0,0],0,0,0]];
ENDMODULE

--- Backups/IRB2400_10kg_1.5m_3/RAPID/TASK1/PROGMOD/MW.mod ---
MODULE MW

    VAR num counter;
    VAR num offsvarX;
    VAR num offsvarY;
    VAR num xoffset;
    VAR num yoffset;
    VAR num pallethole;
    VAR num RunTime:= 5;
    VAR num PinINGripper;
    VAR num Command;
    !REMEMBER TO CHANGE THIS IN FINAL (comment)
    PERS num DMH:= 1;

!Comment While in RobotStudio;
   ! VAR num SignalDelay:= 2;
!Uncomment while in robotstudio:
    !VAR num Din;

  !-------------OWN TARGETS-------------!
  !
  !# TILTED Position of the Pallet from the Home Position (Tilted)
  ! OLD NOT USED CONST robtarget pPalHomeTilt:=[[1015.987042359,-133.981901811,718.978895592],[0.000045049,-0.665857682,-0.00005045,-0.746078778],[-1,-1,-2,0],[9E9,9E9,9E9,9E9,9E9,9E9]];
  !
  ! OLD NOT USED CONST robtarget pPalHomeTilt:=[[1016,-134.1,718.9],[0.00384,-0.59383, -0.00571, -0.80457],[-1,-1,-2,0],[9E9,9E9,9E9,9E9,9E9,9E9]];
  CONST robtarget pPalHomeTilt:=[[1015,-134.1,718.7],[0.00423,-0.5433, -0.0054, -0.8395],[-1,-1,-2,0],[9E9,9E9,9E9,9E9,9E9,9E9]];
!#Position of Slug ready to Drop into HOLE NUMBER 1 of the Pallet on the Conveyer
  CONST robtarget pSlugPallH1D:=[[-306.3,-1341.28,493.07],[0.499794,0.500175,0.500017,-0.500013],[-2,-1,0,0],[9E+09,9E+09,9E+09,9E+09,9E+09,9E+09]];
  !
  !#Position of Slug ready to GRAB PIN IN HOLE NUMBER 1 of the Pallet on the Conveyer

  !Uncomment while in robotstuio: (THIS IS TARGET THAT WORKS WITH SIMULATION)
    CONST robtarget pSlugPallH1G:=[[-306.3,-1341.28,493.07],[0.499794,0.500175,0.500017,-0.500013],[-2,-1,0,0],[9E+09,9E+09,9E+09,9E+09,9E+09,9E+09]];
  !
  !Comment while in robotstuio:(THIS IS THE REAL TARGET)
  !CONST robtarget pSlugPallH1G:=[[-306.3,-1341.28,467.71],[0.499794,0.500175,0.500017,-0.500013],[-2,-1,0,0],[9E+09,9E+09,9E+09,9E+09,9E+09,9E+09]];

!#Position in safe position from conveyor with tilt
	CONST robtarget pConvTilt:=[[-234.5, -1061.8, 596.5], [0.61732, 0.34490, -0.34483, 0.61730],[-2,-1,-2,0],[9E9,9E9,9E9,9E9,9E9,9E9]];

  !New safe position
  CONST robtarget pnewsafe:=[[641.8,420.7,686.3] ,[0.668321,-0.230856,0.668582,0.230329],[0,0,-1,0],[9E+09,9E+09,9E+09,9E+09,9E+09,9E+09]];
  !# SAFE Position of Slug 1 (Eastern Side) on the Dispenser ready to Grip
  ! NOT IN USE CONST robtarget pSlugDispG1Safe:=[[778.35,720.35,650.08],[0.668321,-0.230856,0.668582,0.230329],[0,0,-1,0],[9E+09,9E+09,9E+09,9E+09,9E+09,9E+09]];
  !
CONST robtarget pSlugDispG1Safe:=[[890.6,577.3,657.9],[0.67814,-0.20071,0.678,0.20039],[0,0,-1,0],[9E9,9E9,9E9,9E9,9E9,9E9]];
  !# SAFE Position of Slug 2 (Western Side) on the Dispenser ready to Grip
  !NOT IN USE  CONST robtarget pSlugDispG2Safe:=[[901.56,565.81,651.83],[0.668406,-0.230832,0.668515,0.230301],[0,-1,0,0],[9E+09,9E+09,9E+09,9E+09,9E+09,9E+09]];
  !
CONST robtarget pSlugDispG2Safe:=[[784.1,715.6,657.7],[0.6583,-0.26904,0.65409,0.25768],[0,-1,0,0],[9E9,9E9,9E9,9E9,9E9,9E9]];
  !#INTERMEDIATE Position between dispensers and conveyor
  CONST robtarget pDispConvInt:=[[887.7,-578.4,995.2],[0.65468,0.26515,0.65644,-0.26491],[-1,-1,0,0],[9E9,9E9,9E9,9E9,9E9,9E9]];
  !
 !Position of Slug 1 (Eastern Side) ready to Drop into the Dispenser

  CONST robtarget pSlugDispD1:=[[853,794,1590],[0.668406,-0.230832,0.668515,0.230301],[0,-1,0,0],[9E+09,9E+09,9E+09,9E+09,9E+09,9E+09]];

  !

  !Position of Slug 2 (Western Side) ready to Drop into the Dispenser

  CONST robtarget pSlugDispD2:=[[974,645,1590],[0.668406,-0.230832,0.668515,0.230301],[0,0,-1,0],[9E+09,9E+09,9E+09,9E+09,9E+09,9E+09]];

  !
  !!NEW SAFE TARGETS
  !
   !Safe Position of Slug 1 (Eastern Side) on the Dispenser ready to Grip (150mm from slug)
  CONST robtarget pSafe15DispG1:=[[741.4,686.1,652],[0.668406,-0.230832,0.668515,0.230301],[0,0,-1,0],[9E+09,9E+09,9E+09,9E+09,9E+09,9E+09]];
  !
  !Safe Position of Slug 2 (Western Side) on the Dispenser ready to Grip (150mm from slug)
  CONST robtarget pSafe15DispG2:=[[850.2,551.4,652],[0.668406,-0.230832,0.668515,0.230301],[0,-1,0,0],[9E+09,9E+09,9E+09,9E+09,9E+09,9E+09]];
  !
  !Stop Safe Position of Slug 1 (Eastern Side) on the Dispenser ready to Grip (25mm from slug)
  CONST robtarget pSafe25DispG1:=[[833.2,771,652],[0.668406,-0.230832,0.668515,0.230301],[0,0,-1,0],[9E+09,9E+09,9E+09,9E+09,9E+09,9E+09]];
  !
  !Stop Safe Position of Slug 2 (Western Side) on the Dispenser ready to Grip (25mm from slug)
  CONST robtarget pSafe25DispG2:=[[955,619.4,652],[0.668406,-0.230832,0.668515,0.230301],[0,-1,0,0],[9E+09,9E+09,9E+09,9E+09,9E+09,9E+09]];

  !------------GIVEN TARGETS------------!
  !
  !Position of Slug ready to PickUp from the Centre hole of the Pallet on the Conveyer
  CONST robtarget pSlugPallConvCP:=[[-236.32,-1271.28,467.71],[0.499775,0.500257,0.500025,-0.499943],[-2,-1,0,0],[9E+09,9E+09,9E+09,9E+09,9E+09,9E+09]];
  !
  !Position of Slug ready to Drop into the Centre hole of the Pallet on the Conveyer
  CONST robtarget pSlugPallConvCD:=[[-236.3,-1271.28,493.07],[0.499794,0.500175,0.500017,-0.500013],[-2,-1,0,0],[9E+09,9E+09,9E+09,9E+09,9E+09,9E+09]];
  !
  !Position of Slug 1 (Eastern Side) on the Dispenser ready to Grip
  CONST robtarget pSlugDispG1:=[[851.75,788.07,650.08],[0.668321,-0.230856,0.668582,0.230329],[0,0,-1,0],[9E9,9E9,9E9,9E9,9E9,9E9]];
  !
  !Position of Slug 2 (Western Side) on the Dispenser ready to Grip
  CONST robtarget pSlugDispG2:=[[974.96,633.73,651.83],[0.668406,-0.230832,0.668515,0.230301],[0,-1,0,0],[9E9,9E9,9E9,9E9,9E9,9E9]];
  !
  !Position of the Pallet on the Conveyer
  CONST robtarget pPalletConv:=[[-234.56,-1344.02,396.85],[0.50004,0.499943,-0.50004,0.499977],[-2,-1,-2,0],[9E9,9E9,9E9,9E9,9E9,9E9]];
  !
  !Position of the Pallet in the Home Position
  CONST robtarget pPalletHome:=[[1250.04,-133.95,504.28],[0.000048,-0.707408,-0.000048,-0.706806],[-1,-1,-2,0],[9E9,9E9,9E9,9E9,9E9,9E9]];
  !
  !Calibrate Position for all Joints
  CONST jointtarget jtCalibPos:=[[0,0,0,0,0,0],[9E9,9E9,9E9,9E9,9E9,9E9]];
  !
  !
  !---------TOOL DATA---------!
  !
  !Tool Centre Point (TCP), Orientation, Mass and  COG for the Gripper
  PERS tooldata tGrip:=[TRUE,[[30,0,180],[1,0,0,0]],[1.5,[0,0,80],[1,0,0,0],0,0,0]];
  !
  !Tool Centre Point (TCP), Orientation, Mass and  COG for the Tines
  PERS tooldata tTine:=[TRUE,[[-114.5,0,234.15],[1,0,0,0]],[1.5,[0,0,80],[1,0,0,0],0.04,0.04,0.04]];
  !
  !
  !---------LOAD DATA---------!
  !
  PERS loaddata loSlug:=[0.62,[-35,0,0],[1,0,0,0],0,0,0];
  !
  ! The above code is provided from Steve Kuhle
  !
  !
  !--------PROCEDURES--------!
  !
  !Place pallet on conveyor and return robot to home position or "Waiting position"
  PROC PlacePallet()

   	 MoveJ Offs(pPalletHome,-232,0,100), v1000, z50, tTine;
   	 MoveJ Offs(pPalletHome,-232,0,0), v500, fine, tTine;
     !Moved Pickup position 1 cm)
     MoveL pPalletHome, v200, fine, tTine;
    MoveL Offs(pPalletHome,0,0,50), v200, fine, tTine;
	MoveL pPalHomeTilt, v300, fine, tTine;
    MoveJ Offs(pPalletConv,0,282,200), v1000, z100, tTine;
	MoveL Offs(pPalletConv,0,0,50), v500, fine, tTine;
    MoveL pPalletConv, v200, fine, tTine;
	MoveL Offs(pPalletConv,0,282,0), v200, fine, tTine;

    !if in robotstudio COMMENT:
!    SetGO Dout,255;
!	SetGO \Sdelay := SignalDelay,Dout,0;
TPWrite "Pallet on conveyor";

	MoveL Offs(pPalletConv,0,282,200), v1000, z50, tTine;
	MoveAbsJ jtCalibPos, vMax, fine, tTine;

  ENDPROC

  ! Return pallet to home and return robot to home position or "Waiting position"
PROC ReturnPallet()

    MoveJ Offs(pPalletConv,0,282,200), vMax, fine, tTine;
    MoveL Offs(pPalletConv,0,282,0), v200, fine, tTine;
    MoveL pPalletConv, v200, fine, tTine;
    MoveL Offs(pPalletConv, 0,0,50), v200, fine, tTine; !TILT??
!    MoveJ pConvTilt, v200, fine, tTine;
    MoveJ Offs(pPalletConv,0,282,200), v1000, z100, tTine;
    MoveJ pPalHomeTilt, v1000, z100, tTine;
    MoveJ Offs(pPalletHome,0,0,100), v500, z50, tTine;
    MoveL pPalletHome, v200, fine, tTine;


    MoveL Offs(pPalletHome,-232,0,0), v500, fine, tTine;
    MoveJ Offs(pPalletHome,-232,0,100), v1000, z50, tTine;
    MoveAbsJ jtCalibPos, vMax, fine, tTine;

	!COMMENT if in robotstudio :
!	SetGO Dout,250;
!	SetGO \Sdelay := SignalDelay,Dout,0;
    TPWrite "Pallet returned to table";
ENDPROC


  ! Moves pin to from dispensers to position over pallet center hole pallet.
  PROC GetPin()


    Set Grip;
	WaitTime 1;

	IF Disp1 = 1 THEN
		!Pick pin from dispenser 1 and move to pallet
		TPWrite "Getting pin from dispenser 1";
		!MoveJ pnewsafe, v500, fine, tGrip;
        MoveJ Offs(pSafe15DispG1,-100,-130,200), v1000, z200, tGrip;
		MoveJ pSafe15DispG1, v500, z50, tGrip;

        MoveJ pSafe25DispG1, v500, fine,tGrip;
!        MoveJ pSlugDispG1Safe, v500, fine, tGrip;

		MoveL pSlugDispG1, v200, fine, tGrip;
		Reset Grip;
		WaitTime 1;
		PinINGripper:= 1;

		MoveJ pSafe25DispG1, v500, fine,tGrip;
        MoveJ pSafe15DispG1, v500, z50, tGrip;
        MoveJ Offs(pSafe15DispG1,-100,-130,200), v1000, z200, tGrip;
!        MoveL pSlugDispG1Safe, v200, fine, tGrip;


	ELSEIF Disp2 = 1 THEN
		!Pick pin from dispenser 2 and move to pallet
        TPWrite "Dispenser 1 is empty, getting pin from dispenser 2";
!		MoveJ pSlugDispG2Safe, v1000, fine, tGrip;
        MoveJ Offs(pSafe15DispG2,-100,-130,200), v1000, z200, tGrip;
		MoveJ pSafe15DispG2, v500, z50, tGrip;

        MoveJ pSafe25DispG2, v500, fine,tGrip;
        MoveL pSlugDispG2, v200, fine, tGrip;
		Reset Grip;
		WaitTime 1;
		PinINGripper:= 1;
        MoveJ pSafe25DispG2, v500, fine,tGrip;
        MoveJ pSafe15DispG2, v500, z50, tGrip;
        MoveJ Offs(pSafe15DispG2,-100,-130,200), v1000, z200, tGrip;
!		MoveL pSlugDispG2Safe, v200, fine, tGrip;

	ELSE
		TPWrite "No pin in dispensers";
        RETURN;

		!if in robotstudio COMMENT:
!		SetGO Dout,235;
!		SetGO \Sdelay := SignalDelay,Dout,0;
	ENDIF

	MoveJ pDispConvInt, vMax, z200, tGrip;
	MoveJ Offs(pSlugPallConvCD,0,200,200), v1000, z200, tGrip;
	!MoveJ Offs(pSlugPallConvCD,0,0,200), v1000, fine, tGrip;
ENDPROC




! Calculates the hole and moves the pin from Offs(pSlugPallConvCD,0,0,200) into hole.
!We number the pallet holes from 1 to 25. [and return robot to home position or "Waiting position"??]
PROC DropInPallet()

	!MoveJ Offs(pSlugPallConvCD,0,0,200), v1000, fine, tGrip;
	IF PinINGripper = 1 THEN

    pallethole := Command;
	TPWrite "Hole to be filled: "\Num:=pallethole;
	counter := 0;
	offsvarX := 0;
	offsvarY := 0;

		FOR i FROM 0 TO 4 DO
			FOR j FROM 0 TO 4 DO

			counter := counter + 1;

                IF counter = pallethole THEN
                	offsvarX := i;
			        offsvarY := j;
                ENDIF

			ENDFOR
		ENDFOR

	xoffset := 35*offsvarX;
	yoffset := 35*offsvary;


	TPWrite "X offset from hole 1 = "\ Num:=xoffset;
	TPWrite "Y offset from hole 1 = "\ Num:=yoffset;

	!additional point:
    MoveJ Offs(pSlugPallH1D, xoffset, yoffset, 100), v200, z50, tGrip;
	!
	MoveL Offs(pSlugPallH1D, xoffset, yoffset, 50), v200, fine, tGrip;
	MoveL Offs(pSlugPallH1D, xoffset, yoffset, 0), v200, fine, tGrip;
	Set Grip;
	WaitTime 1;
	PinINGripper:= 0;


	MoveL Offs(pSlugPallH1D, xoffset, yoffset, 100), v200, fine, tGrip;
    MoveJ Offs(pSlugPallConvCD,0,200,200), v1000, fine, tGrip;

!Comment while in robotstudio
!	SetGO Dout,245;
!	SetGO \Sdelay := SignalDelay,Dout,0;


	TPWrite "Slug is placed in pallethole "\Num:=pallethole;

    ENDIF

ENDPROC

!Moves from pallet to homeposition

PROC ToHomePos()
	MoveAbsJ jtCalibPos, v1000, fine, tTine;
ENDPROC

  !Procedure to pick up pin from pallet and return robot to Safe position of pallet
  PROC RemovePin()

      IF PinINGripper = 0 THEN

    pallethole := Command - 100;

    MoveJ Offs(pSlugPallConvCD,0,0,100), v1000, fine, tGrip;
	Set Grip;
	WaitTime 1;

	counter := 0;
	offsvarX := 0;
	offsvarY := 0;

		FOR i FROM 0 TO 4 DO
			FOR j FROM 0 TO 4 DO

			counter := counter + 1;

                IF counter = pallethole THEN
                	offsvarX := i;
			        offsvarY := j;
                ENDIF

			ENDFOR
		ENDFOR

	xoffset := 35*offsvarx;
	yoffset := 35*offsvary;


	TPWrite "X offset from hole 1 = "\ Num:=xoffset;
	TPWrite "Y offset from hole 1 = "\ Num:=yoffset;

	MoveL Offs(pSlugPallH1G, xoffset, yoffset, 100), v200, fine, tGrip;
    MoveL Offs(pSlugPallH1G, xoffset, yoffset, 0), v200, fine, tGrip;
	Reset Grip;
	WaitTime 1;
	PinINGripper:= 1;

	MoveL Offs(pSlugPallH1D, xoffset, yoffset, 100), v200, fine, tGrip;
	MoveL Offs(pSlugPallH1G, xoffset, yoffset, 200), v200, z50, tGrip;
    MoveJ Offs(pSlugPallConvCD,0,200,200), v1000, fine, tGrip;
!Comment while in robotstudio
!SetGO Dout,240;
!SetGO \Sdelay := SignalDelay,Dout,0;
  	TPWrite "Slug is removed from pallethole "\Num:=pallethole;
                ELSE
            TPWrite "Cannot remove pin while pin is in gripper";
      ENDIF

  ENDPROC

PROC InDisp1()
IF PinINGripper = 1 THEN
		MoveAbsJ jtCalibPos, vMax, z200, tGrip;
		MoveL Offs(pSlugDispD1,0,0,10), v1000,fine, tGrip;
		MoveL pSlugDispD1,v200,fine, tGrip;
		Set Grip;
		WaitTime 1;
		PinINGripper:= 0;
		MoveL pSlugDispD1,v200,fine, tGrip;
		MoveL Offs(pSlugDispD1,0,0,10), v1000,fine, tGrip;
		MoveAbsJ jtCalibPos, vMax, fine, tGrip;
		WaitTime 0.5;
		Reset Grip;

		TPWrite "Pin is placed in dispenser 1";
!Comment while in RS
!SetGO Dout,205;
!SetGO \Sdelay := SignalDelay,Dout,0;
ELSE
        TPWrite "No pin in gripper";
ENDIF
ENDPROC

PROC InDisp2()
IF PinINGripper = 1 THEN
		MoveAbsJ jtCalibPos, vMax, z200, tGrip;
		MoveL Offs(pSlugDispD2,0,0,10), v1000,fine, tGrip;
		MoveL pSlugDispD2,v200,fine, tGrip;
		Set Grip;
		PinINGripper:= 0;
		WaitTime 1;
		MoveL pSlugDispD2,v200,fine, tGrip;
		MoveL Offs(pSlugDispD2,0,0,10), v1000,fine, tGrip;
		MoveAbsJ jtCalibPos, vMax, fine, tGrip;
		WaitTime 0.5;
		Reset Grip;
		TPWrite "Pin is placed in dispenser 2";
!Comment while in RS
!SetGO Dout,205;
!SetGO \Sdelay := SignalDelay,Dout,0;
ELSE
        TPWrite "No pin in gripper";
ENDIF

ENDPROC

PROC RunConveyorOUT()
    Reset ConDir;
    Set ConRun;
    SetDO \Sdelay := RunTime, ConRun, 0;
    WaitTime 0.5;

TPWrite "Pallet has been moved out of cell";
!Comment while in RS
!SetGO \Sdelay := RunTime, Dout,225;
!SetGO \Sdelay := SignalDelay,Dout,0;

ENDPROC

PROC RunConveyorIN()
 Set ConDir;
 Set ConRun;
 SetDO \Sdelay := RunTime, ConRun, 0;
 WaitTime 0.5;

TPWrite "Pallet has been moved into cell";
!Comment while in RS
!SetGO \Sdelay := RunTime, Dout,220;
!SetGO \Sdelay := SignalDelay,Dout,0;

ENDPROC
PROC SetPallet()

    MoveJ Offs(pSlugPallConvCD,0,200,200), v1000, z50, tGrip;
    MoveJ Offs(pPalletConv,0,290,100), v200, fine, tTine;
    MoveL Offs(pPalletConv,0,290,0), v200, fine, tTine;
    MoveL Offs(pPalletConv,0,-100,0), v200, fine, tTine;
    MoveL Offs(pPalletConv, 0,-100,50), v200, fine, tTine;
    MoveL pConvTilt, v200, fine, tTine;
    MoveL Offs(pPalletConv, 0,0,50), v200, fine, tTine;
    MoveL pPalletConv, v200, fine, tTine;
    MoveL Offs(pPalletConv, 0,282,0), v200, fine, tTine;
    MoveJ Offs(pSlugPallConvCD,0,200,200), v1000, fine, tGrip;

    TPWrite "Pallet has been reset on conveyor";
   !Comment while in RS
!    SetGO Dout,215;
!    SetGO \Sdelay := SignalDelay,Dout,0;
ENDPROC
!--------MAIN PROCEDURE--------!
  PROC main()
!Comment while in RS
!   WaitDI Din, 0;      !Do not start program before Din = zero
!   SetGO Dout,210;     !Tell vision program is running
!   SetGO \Sdelay := SignalDelay,Dout,0;
!   WaitTime 0.5;       !To give system some time

!Unomment while in robotstudio
     WaitDI All_OK, 0; !For simulating "WaitDI Din, 0; !Do not start program before Din = zero"


    Reset Grip;         !Closing grip before starting
    Reset ConRun;       !Make sure the conveyor does not run
    PinINGripper:= 0;

WHILE DMH = 1 DO

!Comment while in robotstudio:
!        Command:= Din;
!Unomment while in robotstudio:
        TPReadNum Command, "Set digital input?";

!#Procedure for placing pallet on conveyor
IF Command = 200 THEN
		PlacePallet;
ENDIF

!#Procedure for returning pallet to table
IF Command = 222 THEN
		ReturnPallet;
ENDIF

!#Procedure for placing pin in pallet and return to safe position pallet.
! If no pin in gripper it picks from dispenser. Oterwise it places current pin in hole
IF Command > 0 AND Command <=25  THEN

        IF PinINGripper = 1 THEN
				DropInPallet;
        ELSEIF PinINGripper = 0 THEN
				GetPin;
				DropInPallet;
        ENDIF
ENDIF

!#Procedure for picking pin from pallet and return to safe position pallet
IF Command > 100 AND Command <=125 THEN
			RemovePin;
ENDIF

!#Procedure for returning robot to home, if pin in gripper->Drop it in Disp1.
IF Command = 26 THEN
    IF PinINGripper = 1 THEN
		InDisp1;
	ENDIF
        ToHomePos;
		Reset Grip;
ENDIF

!#Procedure for running conveyor OUT of cell
IF Command = 27 THEN
            RunConveyorOUT;
ENDIF

!#Procedure for running conveyor INTO cell
IF Command = 28 THEN
		RunConveyorIN;
ENDIF

!#Procedure for reseting the pallet on conveyor. Picks up and places
IF Command = 29 THEN
		SetPallet;
ENDIF
!#Procedure for placing pin in dispenser 1
 IF Command = 126 THEN
        InDisp1;
ENDIF

!#Procedure for placing pin in dispenser 2
IF Command = 127 THEN
           InDisp2;
ENDIF


WaitTime 1;     !To make sure the loop doesnt run too fast

    ENDWHILE

    TPWrite "Program is stopped because something is wrong!";
    !Comment while in RS
!    SetGO Dout,230;
!    SetGO \Sdelay := SignalDelay,Dout,0;
  ENDPROC

ENDMODULE

--- Backups/IRB2400_10kg_1.5m_3/SYSPAR/EIO.cfg ---
EIO:CFG_1.0:5:0::
#
EIO_BUS:

      -Name "Virtual1" -ConnectorID "SIM1"
#
EIO_UNIT_TYPE:

      -Name "Virtual" -VendorName "ABB" -ProductName "Virtual unit"
#
EIO_UNIT:

      -Name "MyBus" -UnitType "Virtual" -Bus "Virtual1" -TrustLevel 0
#
EIO_SIGNAL:

      -Name "Grip" -SignalType "DO" -Unit "MyBus" -UnitMap "1" -Access "Default"

      -Name "Disp1" -SignalType "DI" -Unit "MyBus" -UnitMap "2"\
      -Access "Default"

      -Name "Disp2" -SignalType "DI" -Unit "MyBus" -UnitMap "3"\
      -Access "Default"

      -Name "ConDir" -SignalType "DO" -Unit "MyBus" -UnitMap "4"\
      -Access "Default"

      -Name "ConRun" -SignalType "DO" -Unit "MyBus" -UnitMap " 3"\
      -Access "Default"

      -Name "All_OK" -SignalType "DI" -Unit "MyBus" -UnitMap "4"\
      -Access "Default"

      -Name "NewPinInDispenser" -SignalType "DI" -Unit "MyBus" -UnitMap "5"\
      -Access "Default"
#
EIO_ACCESS:

      -Name "All" -Rapid  -LocalManual  -LocalAuto  -RemoteManual  -RemoteAuto
